{attribute 'TcGenerated'}
{attribute 'no-analysis'}
{attribute 'linkalways'}
// This function has been automatically generated from the project information.
VAR_GLOBAL CONSTANT
	{attribute 'const_non_replaced'}
	stLibVersion_Tc3_Event : ST_LibVersion := (iMajor := 0, iMinor := 0, iBuild := 0, iRevision := 7, nFlags := 0, sVersion := '0.0.0.7');
END_VAR

(* stored: Version 1.1.0.1
   GVL Global_Version: Id {743ce783-7fa5-4f64-8ad9-9ec7d60dfe93} *)
